TYPE RemoteData :
STRUCT
	// Feedback data sendt from PLC to UDP interface
	Tx		: RemoteDataTx;
	// Data recieved from UDP interface to PLC
	Rx		: RemoteDataRx;
END_STRUCT
END_TYPE

(* stored: Version 1.1.0.1, ProductVersion 3.1.4020.12
   DUT RemoteData: Id {0afe537a-cf1d-4220-8de7-7cc910cf92e8} *)
